(* CODESYS project PropertiesExport.export

Project tree, tasks and I/O mapping:
  program Main [ST]
  function block Motor [ST]: IsRunning
*)

// Main
PROGRAM Main
VAR_INPUT
	MotorA : Motor;
END_VAR
VAR
	MotorAIsRunning : BOOL;
END_VAR


// Set property
MotorA.IsRunning := TRUE;


// Get property
MotorAIsRunning := MotorA.IsRunning;

END_PROGRAM

// Motor
FUNCTION_BLOCK Motor
VAR
	_isRunning : BOOL;
END_VAR

PROPERTY PUBLIC IsRunning : BOOL
GET

// Perform validation if necessary

IsRunning := _isRunning;
END_GET
SET

// Perform validation if necessary

_isRunning := IsRunning;
END_SET
END_PROPERTY

END_FUNCTION_BLOCK
